{attribute addProperty BoxType "AT2050-0501-0019"}
{attribute addProperty Id "A_0081_AT2002_5250_0018_AT2002_5250AT2002_3DCFC8D064080"}
{attribute addProperty CRC "862273250"}
{attribute addProperty SizeInBites "640"}
{attribute addProperty SizeInBytes "80"}
TYPE A_0069_AT2050_0501_0019_AT2050_0501_33653EE2 EXTENDS AT2050_9506A482 :
STRUCT
	{attribute addProperty Name "A_0081_AT2002_5250_0018_AT2002_5250"}
	A_0081_AT2002_5250_0018_AT2002_5250 : AT2002_3DCFC8D0;
END_STRUCT
END_TYPE

(* stored: Version 1.2.0.0, ProductVersion 3.1.4024.9
   DUT A_0069_AT2050_0501_0019_AT2050_0501_33653EE2: Id {2a41fc50-19d8-478c-acb3-7ac4f8f543e6} *)
